FUNCTION_BLOCK TIME2REAL (* Basic Function Block Type *)
  (* Standard: 61499-2 *)
  (* Version 0.0, 6/13/2026, Schneider Electric, Template *)
  PACKAGE SE.Nereda;
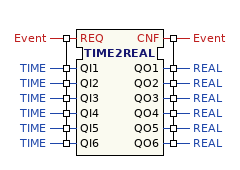
  EVENT_INPUT
    REQ WITH QI1, QI2, QI3, QI4, QI5, QI6; (* Normal Execution Request *)
  END_EVENT
  EVENT_OUTPUT
    CNF WITH QO1, QO2, QO3, QO4, QO5, QO6; (* Execution Confirmation *)
  END_EVENT
  VAR_INPUT
    QI1 : TIME; (* Input event qualifier *)
    QI2 : TIME;
    QI3 : TIME;
    QI4 : TIME;
    QI5 : TIME;
    QI6 : TIME;
  END_VAR
  VAR_OUTPUT
    QO1 : REAL; (* Output event qualifier *)
    QO2 : REAL;
    QO3 : REAL;
    QO4 : REAL;
    QO5 : REAL;
    QO6 : REAL;
  END_VAR
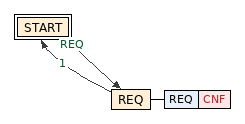
  EC_STATES
    START; (* Initial State *)
    REQ : REQ -> CNF; (* Normal execution *)
  END_STATES
  EC_TRANSITIONS
    START TO REQ := REQ;
    REQ TO START := 1;
  END_TRANSITIONS
  ALGORITHM REQ IN ST: (* Normally executed algorithm *)
;
QO1 := TIME_TO_REAL(QI1/1000);
QO2 := TIME_TO_REAL(QI2/1000);
QO3 := TIME_TO_REAL(QI3/1000);
QO4 := TIME_TO_REAL(QI4/1000);
QO5 := TIME_TO_REAL(QI5/1000);
QO6 := TIME_TO_REAL(QI6/1000);
  END_ALGORITHM
END_FUNCTION_BLOCK
